Staubli VAL3: checkTrackArea.pgx

program checkTrackArea(num x_nConvNum (dimensions=1), tool x_tActivTool (dimensions=1), num& x_nArea[] (dimensions=1))
begin
  switch x_nConvNum
    case 0
      call cnv0:checkTrackArea(x_tActivTool,x_nArea)
    break
    case 1
      call cnv1:checkTrackArea(x_tActivTool,x_nArea)
    break
    default
      x_nArea=-1
    break
  endSwitch
end
